// TIA Portal project "three-phase motor" (V15)

(* hardware
DEVICE "S7-1200 station_1"  S7-1200 Station
   slot 0: "Rack_0"  S7-1200 Rack  Rack  V1.0
   slot 1: "PLC_1"  CPU 1214C AC/DC/Rly  6ES7 214-1BG40-0XB0  V4.2
*)

// ===== PLC "PLC_1"  CPU 1214C AC/DC/Rly =====

VAR_GLOBAL   // PLC tag table "COLUMN DRILL WHIO"
   "ESO" AT %I0.0 : Bool;   // EM STOP (NC)
   "S1" AT %I0.2 : Bool;   // STOP (NC)
   "S2" AT %I0.3 : Bool;   // START (NO)
   "P1" AT %Q0.0 : Bool;   // READY (G) 24VDC
   "P2" AT %Q0.1 : Bool;   // MOTOR ON (Y) 24VDC
   "P3" AT %Q0.2 : Bool;   // MALF (R) 24VDC
   "F3" AT %I0.1 : Bool;   // OVERLOAD (NC)
   "Q2" AT %Q0.5 : Bool;   // MOTOR CONTACTOR 240VDC
END_VAR

ORGANIZATION_BLOCK "Main"   // OB1, LAD, ProgramCycle
TITLE = "Main Program Sweep (Cycle)"
{ S7_Optimized_Access := 'TRUE' }
VERSION : 0.1
   VAR_INPUT
      Initial_Call : Bool;   // Initial call of this OB
      Remanence : Bool;   // =True, if remanent data are available
   END_VAR
BEGIN

REGION Network 1: READY (G) 24VDC
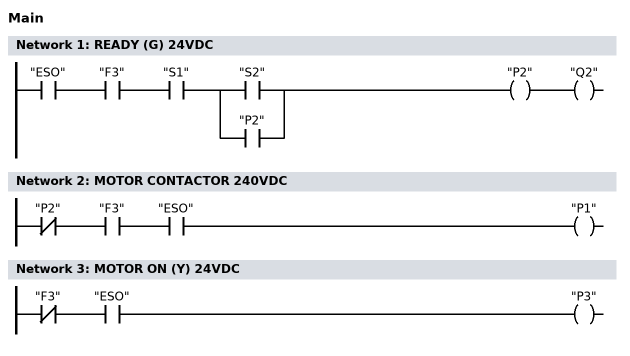
   RUNG wire#powerrail
      Contact( "ESO" )
      Contact( "F3" )
      Contact( "S1" )
      wire#w1
      Contact( "S2" )
      wire#w2
      Coil( "P2" )
      Coil( "Q2" )
   END_RUNG
   RUNG wire#w1
      Contact( "P2" )
   END_RUNG wire#w2
   // the same network as SCL:
   "P2" := "ESO" AND "F3" AND "S1" AND ("S2" OR "P2");
   "Q2" := "P2";
END_REGION

REGION Network 2: MOTOR CONTACTOR 240VDC
   RUNG wire#powerrail
      I_Contact( "P2" )
      Contact( "F3" )
      Contact( "ESO" )
      Coil( "P1" )
   END_RUNG
   // the same network as SCL:
   "P1" := NOT "P2" AND "F3" AND "ESO";
END_REGION

REGION Network 3: MOTOR ON (Y) 24VDC
   RUNG wire#powerrail
      I_Contact( "F3" )
      Contact( "ESO" )
      Coil( "P3" )
   END_RUNG
   // the same network as SCL:
   "P3" := NOT "F3" AND "ESO";
END_REGION
END_ORGANIZATION_BLOCK